FUNCTION_BLOCK WrappedComponentExample EXTENDS TcoCore.TcoComponent
VAR_OUTPUT
END_VAR
VAR
    _config : WrappedComponentExample_Config;
    _status : WrappedComponentExample_Status;
    _control : WrappedComponentExample_Control;
    _components : WrappedComponentsExample := (Parent := THIS^);
    _throwTask : TcoCore.TcoTask(THIS^);
    _restoreTask : TcoCore.TcoTask(THIS^);
END_VAR

PROPERTY Components : REFERENCE TO WrappedComponentsExample
GET
Components ref= _components;
END_GET
END_PROPERTY

(*~
    <docu>
        <summary>
            Restores this instance to the Ready state. Can be called explicitly or from within one of the restore mechanisms.
        </summary>
    </docu>
~*)
METHOD Restore : ITcoRestorable
END_METHOD

(*~
    <docu>
        <summary>
            Custom service (manual, maintenance) logic.
            This method must be implemented in derived class.
        </summary>
    </docu>
~*)
METHOD PROTECTED ServiceMode
END_METHOD

END_FUNCTION_BLOCK

(* stored: Version 1.1.0.1, ProductVersion 3.1.4024.12
   POU WrappedComponentExample: Id {47c5ed63-a639-0668-2732-bb135eb269d1}, SpecialFunc None
   Property Components: Id {93c570c0-6fde-096d-1d23-f4f966fbd389}
   Get Get: Id {2f61461f-0e40-0651-14cf-7108bc9b05d2}
   Method Restore: Id {07efd12a-84ef-01eb-0654-21e61fba155a}
   Method ServiceMode: Id {cb7697df-4f59-092b-27b8-f175ac230c09} *)
